ABB RAPID module: 000392E8

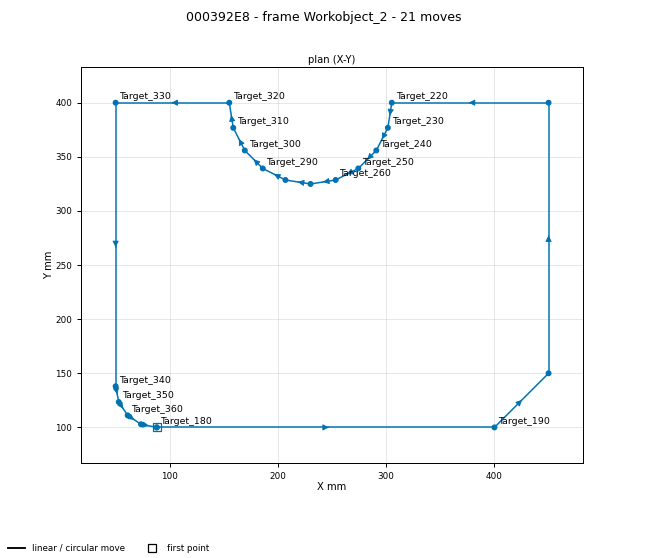
[picture p0: tool path of 000392E8 in frame Workobject_2, 21 of 38 moves have a stored position in this frame; points joined in program order, loops and branches not executed]
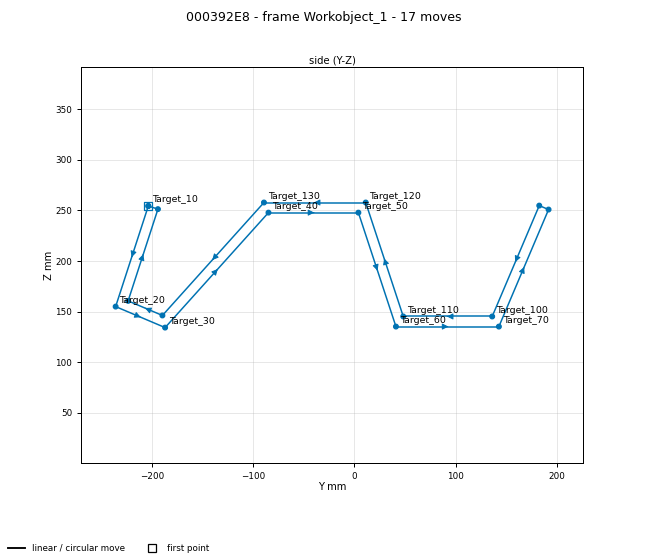
[picture p1: tool path of 000392E8 in frame Workobject_1, 17 of 38 moves have a stored position in this frame; points joined in program order, loops and branches not executed]
MODULE Module1
        CONST robtarget Target_10:=[[-60,-203.867068409,254.436574641],[0.11061582,0.698407699,0.110615923,0.698394548],[0,0,0,0],[9E+09,9E+09,9E+09,9E+09,9E+09,9E+09]];
    CONST robtarget Target_20:=[[-59.999999999,-236.184577372,154.97350934],[0.11061582,0.698407699,0.110615923,0.698394548],[0,0,0,0],[9E+09,9E+09,9E+09,9E+09,9E+09,9E+09]];
    CONST robtarget Target_30:=[[-60,-187.258965467,134.205819219],[0.11061582,0.698407699,0.110615923,0.698394548],[0,0,0,0],[9E+09,9E+09,9E+09,9E+09,9E+09,9E+09]];
    CONST robtarget Target_40:=[[-60,-85.044509222,247.891489668],[0.11061582,0.698407699,0.110615923,0.698394548],[0,0,0,0],[9E+09,9E+09,9E+09,9E+09,9E+09,9E+09]];
    CONST robtarget Target_50:=[[-59.999999999,3.878988935,247.891489668],[0.11061582,0.698407699,0.110615923,0.698394548],[0,0,0,0],[9E+09,9E+09,9E+09,9E+09,9E+09,9E+09]];
    CONST robtarget Target_60:=[[-60,41.014913739,135.202937257],[0.11061582,0.698407699,0.110615923,0.698394548],[0,0,0,0],[9E+09,9E+09,9E+09,9E+09,9E+09,9E+09]];
    CONST robtarget Target_70:=[[-60,142.810926639,135.202937257],[0.11061582,0.698407699,0.110615923,0.698394548],[0,0,0,0],[9E+09,9E+09,9E+09,9E+09,9E+09,9E+09]];
    CONST robtarget Target_80:=[[-60,191.937475674,250.937834026],[0.11061582,0.698407699,0.110615923,0.698394548],[0,0,0,0],[9E+09,9E+09,9E+09,9E+09,9E+09,9E+09]];
    CONST robtarget Target_90:=[[-60.000000001,182.732427139,254.845145311],[0.11061582,0.698407699,0.110615923,0.698394548],[0,0,0,0],[9E+09,9E+09,9E+09,9E+09,9E+09,9E+09]];
    CONST robtarget Target_100:=[[-60,136.192071026,145.202937257],[0.11061582,0.698407699,0.110615923,0.698394548],[0,0,0,0],[9E+09,9E+09,9E+09,9E+09,9E+09,9E+09]];
    CONST robtarget Target_110:=[[-60,48.248472324,145.202937257],[0.11061582,0.698407699,0.110615923,0.698394548],[0,0,0,0],[9E+09,9E+09,9E+09,9E+09,9E+09,9E+09]];
    CONST robtarget Target_120:=[[-60,11.112547519,257.891489669],[0.11061582,0.698407699,0.110615923,0.698394548],[0,0,0,0],[9E+09,9E+09,9E+09,9E+09,9E+09,9E+09]];
    CONST robtarget Target_130:=[[-60.000000001,-89.501123873,257.891489669],[0.11061582,0.698407699,0.110615923,0.698394548],[0,0,0,0],[9E+09,9E+09,9E+09,9E+09,9E+09,9E+09]];
    CONST robtarget Target_140:=[[-60,-189.92256825,146.200055295],[0.11061582,0.698407699,0.110615923,0.698394548],[0,0,0,0],[9E+09,9E+09,9E+09,9E+09,9E+09,9E+09]];
    CONST robtarget Target_150:=[[-60,-223.842393157,160.598166739],[0.11061582,0.698407699,0.110615923,0.698394548],[0,0,0,0],[9E+09,9E+09,9E+09,9E+09,9E+09,9E+09]];
    CONST robtarget Target_160:=[[-60,-194.356503245,251.346404697],[0.11061582,0.698407699,0.110615923,0.698394548],[0,0,0,0],[9E+09,9E+09,9E+09,9E+09,9E+09,9E+09]];
    CONST robtarget Target_170:=[[-60,-203.867068409,254.436574641],[0.11061582,0.698407699,0.110615923,0.698394548],[0,0,0,0],[9E+09,9E+09,9E+09,9E+09,9E+09,9E+09]];
    CONST robtarget Target_180:=[[88.000388799,99.999868845,104.132758068],[0,0,1,0],[0,0,0,0],[9E+09,9E+09,9E+09,9E+09,9E+09,9E+09]];
    CONST robtarget Target_190:=[[400.000388799,99.999868845,104.132758068],[0,0,1,0],[0,0,0,0],[9E+09,9E+09,9E+09,9E+09,9E+09,9E+09]];
    CONST robtarget Target_200:=[[450.000388799,149.999868845,104.132758068],[0,0,1,0],[0,0,0,0],[9E+09,9E+09,9E+09,9E+09,9E+09,9E+09]];
    CONST robtarget Target_210:=[[450.000388799,399.999868845,104.132758068],[0,0,1,0],[0,0,0,0],[9E+09,9E+09,9E+09,9E+09,9E+09,9E+09]];
    CONST robtarget Target_220:=[[305.168957026,399.999868845,104.132758068],[0,0,1,0],[0,0,0,0],[9E+09,9E+09,9E+09,9E+09,9E+09,9E+09]];
    CONST robtarget Target_230:=[[301.49407059,376.797549043,104.132758068],[0,0,1,0],[0,0,0,0],[9E+09,9E+09,9E+09,9E+09,9E+09,9E+09]];
    CONST robtarget Target_240:=[[290.829134771,355.866433964,104.132758068],[0,0,1,0],[0,0,0,0],[9E+09,9E+09,9E+09,9E+09,9E+09,9E+09]];
    CONST robtarget Target_250:=[[274.218107793,339.255406986,104.132758068],[0,0,1,0],[0,0,0,0],[9E+09,9E+09,9E+09,9E+09,9E+09,9E+09]];
    CONST robtarget Target_260:=[[253.286992714,328.590471167,104.132758068],[0,0,1,0],[0,0,0,0],[9E+09,9E+09,9E+09,9E+09,9E+09,9E+09]];
    CONST robtarget Target_270:=[[230.084672912,324.915584731,104.132758068],[0,0,1,0],[0,0,0,0],[9E+09,9E+09,9E+09,9E+09,9E+09,9E+09]];
    CONST robtarget Target_280:=[[206.882353111,328.590471167,104.132758068],[0,0,1,0],[0,0,0,0],[9E+09,9E+09,9E+09,9E+09,9E+09,9E+09]];
    CONST robtarget Target_290:=[[185.951238032,339.255406986,104.132758068],[0,0,1,0],[0,0,0,0],[9E+09,9E+09,9E+09,9E+09,9E+09,9E+09]];
    CONST robtarget Target_300:=[[169.340211054,355.866433964,104.132758068],[0,0,1,0],[0,0,0,0],[9E+09,9E+09,9E+09,9E+09,9E+09,9E+09]];
    CONST robtarget Target_310:=[[158.675275235,376.797549043,104.132758068],[0,0,1,0],[0,0,0,0],[9E+09,9E+09,9E+09,9E+09,9E+09,9E+09]];
    CONST robtarget Target_320:=[[155.000388799,399.999868845,104.132758068],[0,0,1,0],[0,0,0,0],[9E+09,9E+09,9E+09,9E+09,9E+09,9E+09]];
    CONST robtarget Target_330:=[[50.000388799,399.999868845,104.132758068],[0,0,1,0],[0,0,0,0],[9E+09,9E+09,9E+09,9E+09,9E+09,9E+09]];
    CONST robtarget Target_340:=[[50.000388799,137.999868845,104.132758068],[0,0,1,0],[0,0,0,0],[9E+09,9E+09,9E+09,9E+09,9E+09,9E+09]];
    CONST robtarget Target_350:=[[52.892966564,123.457898415,104.132758068],[0,0,1,0],[0,0,0,0],[9E+09,9E+09,9E+09,9E+09,9E+09,9E+09]];
    CONST robtarget Target_360:=[[61.130331114,111.12981116,104.132758068],[0,0,1,0],[0,0,0,0],[9E+09,9E+09,9E+09,9E+09,9E+09,9E+09]];
    CONST robtarget Target_370:=[[73.458418369,102.892446609,104.132758068],[0,0,1,0],[0,0,0,0],[9E+09,9E+09,9E+09,9E+09,9E+09,9E+09]];
    CONST robtarget Target_380:=[[88.000388799,99.999868845,104.132758068],[0,0,1,0],[0,0,0,0],[9E+09,9E+09,9E+09,9E+09,9E+09,9E+09]];
!***********************************************************
    !
    ! Module:  Module1
    !
    ! Description:
    !   <Insert description here>
    !
    ! Author: user
    !
    ! Version: 1.0
    !
    !***********************************************************


    !***********************************************************
    !
    ! Procedure main
    !
    !   This is the entry point of your program
    !
    !***********************************************************
    PROC main()
        !Add your code here
    ENDPROC
    PROC Path_10()
        MoveL Target_10,v1000,z100,MyTool\WObj:=Workobject_1;
        MoveL Target_20,v1000,z100,MyTool\WObj:=Workobject_1;
        MoveL Target_30,v1000,z100,MyTool\WObj:=Workobject_1;
        MoveL Target_40,v1000,z100,MyTool\WObj:=Workobject_1;
        MoveL Target_50,v1000,z100,MyTool\WObj:=Workobject_1;
        MoveL Target_60,v1000,z100,MyTool\WObj:=Workobject_1;
        MoveL Target_70,v1000,z100,MyTool\WObj:=Workobject_1;
        MoveL Target_80,v1000,z100,MyTool\WObj:=Workobject_1;
        MoveL Target_90,v1000,z100,MyTool\WObj:=Workobject_1;
        MoveL Target_100,v1000,z100,MyTool\WObj:=Workobject_1;
        MoveL Target_110,v1000,z100,MyTool\WObj:=Workobject_1;
        MoveL Target_120,v1000,z100,MyTool\WObj:=Workobject_1;
        MoveL Target_130,v1000,z100,MyTool\WObj:=Workobject_1;
        MoveL Target_140,v1000,z100,MyTool\WObj:=Workobject_1;
        MoveL Target_150,v1000,z100,MyTool\WObj:=Workobject_1;
        MoveL Target_160,v1000,z100,MyTool\WObj:=Workobject_1;
        MoveL Target_170,v1000,z100,MyTool\WObj:=Workobject_1;
    ENDPROC
    PROC Path_20()
        MoveL Target_180,v1000,z100,MyTool\WObj:=Workobject_2;
        MoveL Target_190,v1000,z100,MyTool\WObj:=Workobject_2;
        MoveL Target_200,v1000,z100,MyTool\WObj:=Workobject_2;
        MoveL Target_210,v1000,z100,MyTool\WObj:=Workobject_2;
        MoveL Target_220,v1000,z100,MyTool\WObj:=Workobject_2;
        MoveL Target_230,v1000,z100,MyTool\WObj:=Workobject_2;
        MoveL Target_240,v1000,z100,MyTool\WObj:=Workobject_2;
        MoveL Target_250,v1000,z100,MyTool\WObj:=Workobject_2;
        MoveL Target_260,v1000,z100,MyTool\WObj:=Workobject_2;
        MoveL Target_270,v1000,z100,MyTool\WObj:=Workobject_2;
        MoveL Target_280,v1000,z100,MyTool\WObj:=Workobject_2;
        MoveL Target_290,v1000,z100,MyTool\WObj:=Workobject_2;
        MoveL Target_300,v1000,z100,MyTool\WObj:=Workobject_2;
        MoveL Target_310,v1000,z100,MyTool\WObj:=Workobject_2;
        MoveL Target_320,v1000,z100,MyTool\WObj:=Workobject_2;
        MoveL Target_330,v1000,z100,MyTool\WObj:=Workobject_2;
        MoveL Target_340,v1000,z100,MyTool\WObj:=Workobject_2;
        MoveL Target_350,v1000,z100,MyTool\WObj:=Workobject_2;
        MoveL Target_360,v1000,z100,MyTool\WObj:=Workobject_2;
        MoveL Target_370,v1000,z100,MyTool\WObj:=Workobject_2;
        MoveL Target_380,v1000,z100,MyTool\WObj:=Workobject_2;
    ENDPROC
ENDMODULE
